(* IEC 61131-3 sources: LEAP-JSS-Paper1-Artifact/software/LEAP/data/demo/sample_project, 1 file *)

(* ---- lc_kpi.st ---- *)
// KPI: SOx Emissions Concentration (kg/m3)
VAR
    soxConc : REAL := 0.0;
    soxMassFlow : REAL := 0.0;
    volFlow : REAL := 0.0;
END_VAR

(* Example structured text placeholder *)
soxConc := 15.2; (* pretend this comes from an analyzer tag *)
soxMassFlow := 233.4;
volFlow := 15.3;
